// Mitsubishi GX Works2 project: tutor01_ladder   PLC: FX1N/FX1NC

PROGRAM MAIN
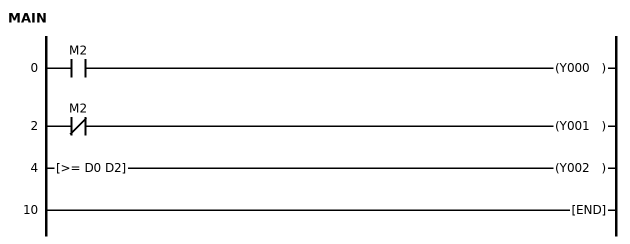
0     LD      M2
      OUT     Y000
2     LDI     M2
      OUT     Y001
4     LD>=    D0 D2
      OUT     Y002
10    END
END_PROGRAM
